TYPE Item :
STRUCT
	Id: UDINT := 0;
	Recipe: Recipe;
END_STRUCT
END_TYPE

(* stored: Version 1.1.0.1, ProductVersion 3.1.4024.12
   DUT Item: Id {69da64a5-f945-4cdb-8879-8319da478ca9} *)
